Omron CX-Programmer project NewProject (CX-Programmer 9.75)

# PLC Timer: CP1E N30

## Global symbols (name address type ; comment)
T000 BOOL  ; T0

## Program NewProgram1 (cyclic task 0)
Local symbols
Lamp1 100.01 BOOL
Lamp2 100.02 BOOL
Lamp3 100.03 BOOL
Lamp4 100.04 BOOL
MainSupply 100.00 BOOL
START 0.00 BOOL
STOP 0.01 BOOL
Sw1 0.02 BOOL
TIM 0.00 BOOL

### Section Section1

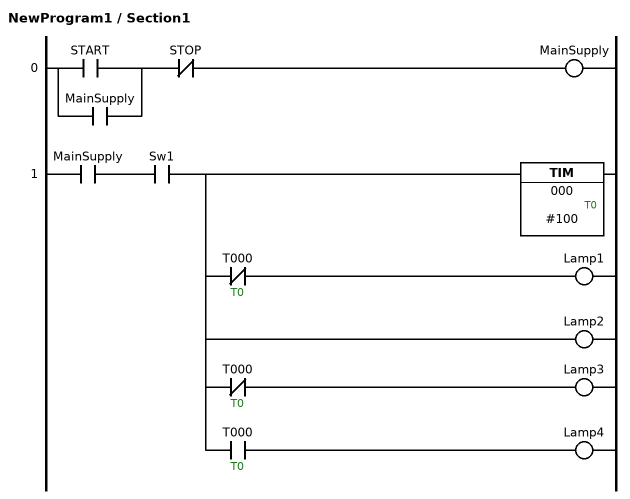
; rung 0
LD START
OR MainSupply
ANDNOT STOP
OUT MainSupply
; rung 1
LD MainSupply
AND Sw1
OUT TR0
TIM 000 #100  ; T0
ANDNOT T000  ; T0
OUT Lamp1
LD TR0
OUT Lamp2
ANDNOT T000  ; T0
OUT Lamp3
LD TR0
AND T000  ; T0
OUT Lamp4

### Section END
; rung 0
END(001)